SUBAPPLICATION Uebung_016c_AX (* Background Colour umschalten -- mit SubApp für SEL und INITVAL *)
  (* Standard: 61499-2; Description: Copyright (c) 2026 Meisterschulen am Ostbahnhof This program and the accompanying materials are made available under the terms of the Eclipse Public License 2.0 which is available at https://www.eclipse.org/legal/epl-2.0/ SPDX-License-Identifier: EPL-2.0 *)
  (* Version 1.0, 2026-09-10, Franz Höpfinger, Meisterschulen am Ostbahnhof, initial API and implementation and/or initial documentation *)
  PACKAGE Uebungen;
  IMPORT isobus::UT::io::Softkey::SoftKeyActivationCode::SK_RELEASED;
  IMPORT Uebungen::const::UT::DefaultPool::SoftKey_F1;
  IMPORT Uebungen::const::UT::DefaultPool::SoftKey_F2;
  IMPORT Uebungen::const::UT::DefaultPool::SoftKey_F7;
  IMPORT isobus::UT::Q::const::colours::COLOR_GREEN;
  IMPORT isobus::UT::Q::const::colours::COLOR_WHITE;
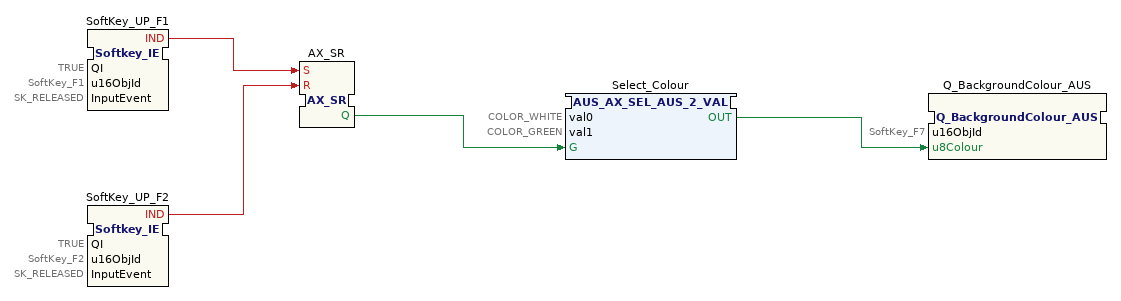
  FBS
    SoftKey_UP_F1 : isobus::UT::io::Softkey::Softkey_IE(QI := TRUE, u16ObjId := SoftKey_F1, InputEvent := SK_RELEASED);
    SoftKey_UP_F2 : isobus::UT::io::Softkey::Softkey_IE(QI := TRUE, u16ObjId := SoftKey_F2, InputEvent := SK_RELEASED);
    AX_SR : adapter::events::unidirectional::AX_SR;
    Q_BackgroundColour_AUS : isobus::UT::Q::Q_BackgroundColour_AUS(u16ObjId := SoftKey_F7);
  END_FBS
  SUBAPPS
    Select_Colour : MyLib::sys::AUS_AX_SEL_AUS_2_VAL(val0 := COLOR_WHITE, val1 := COLOR_GREEN);
  END_SUBAPPS
  EVENT_CONNECTIONS
    SoftKey_UP_F1.IND TO AX_SR.S;
    SoftKey_UP_F2.IND TO AX_SR.R;
  END_CONNECTIONS
  ADAPTER_CONNECTIONS
    AX_SR.Q TO Select_Colour.G;
    Select_Colour.OUT TO Q_BackgroundColour_AUS.u8Colour;
  END_CONNECTIONS
END_SUBAPPLICATION
